# EPICS autosave request: iocs/pvxsDriverIOC/iocBoot/iocPvaDriver/auto_settings.req
file "pvxsDriver_settings.req",      P=$(P),  R=cam1:
file "NDStdArrays_settings.req",    P=$(P),  R=image1:
file "commonPlugin_settings.req",   P=$(P)
